FUNCTION_BLOCK NeredaSludgeBuffer_2_HMI (* Service Interface Function Block Type *)
  (* Standard: 61499-2 *)
  (* Version 0.0, 4/25/2024, SESA713705, Schneider Electric, template *)
  PACKAGE SE.Nereda;
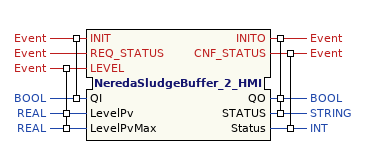
  EVENT_INPUT
    INIT WITH QI;
    REQ_STATUS;
    LEVEL WITH LevelPv, LevelPvMax;
  END_EVENT
  EVENT_OUTPUT
    INITO WITH QO, STATUS;
    CNF_STATUS WITH Status;
  END_EVENT
  VAR_INPUT
    QI : BOOL;
    LevelPv : REAL;
    LevelPvMax : REAL;
  END_VAR
  VAR_OUTPUT
    QO : BOOL; (* Event Output Qualifier *)
    STATUS : STRING; (* Service Status *)
    Status : INT;
  END_VAR
  SERVICE /
    SEQUENCE 
    END_SEQUENCE
  END_SERVICE
END_FUNCTION_BLOCK
